FUNCTION_BLOCK MockEventHandler IMPLEMENTS I_EventHandler
VAR
	_eventsHandled : INT;
	_lastEventHandled : I_Event;
END_VAR

PROPERTY EventsHandled : int
GET
EventsHandled := _eventsHandled;
END_GET
END_PROPERTY

METHOD HandleEvent
VAR_INPUT
	Event	: I_Event;
END_VAR
_eventsHandled := _eventsHandled + 1;
_lastEventHandled := Event;
END_METHOD

PROPERTY PUBLIC LastEventHandled : I_Event
GET
END_GET
END_PROPERTY

END_FUNCTION_BLOCK

(* stored: Version 1.1.0.1, ProductVersion 3.1.4024.12
   POU MockEventHandler: Id {58a62b4e-121a-499d-9f9c-e292ae4280ba}, SpecialFunc None
   Property EventsHandled: Id {ffaf055a-5ff2-4cf4-9302-3d63054b5abf}
   Get Get: Id {581825b6-ffe5-426e-ab27-85efbc5d8312}
   Method HandleEvent: Id {638fbefe-5ea6-4f53-b032-9046544ae9f1}
   Property LastEventHandled: Id {a257476f-6192-4d09-a8c9-08d67b6b10f4}
   Get Get: Id {babb7d60-9682-45bc-9954-9421a7735d40} *)
